// Mitsubishi GX Works2 project: PLC 특수기능 (래치 릴레이)   PLC: Q03UDV

PROGRAM MAIN
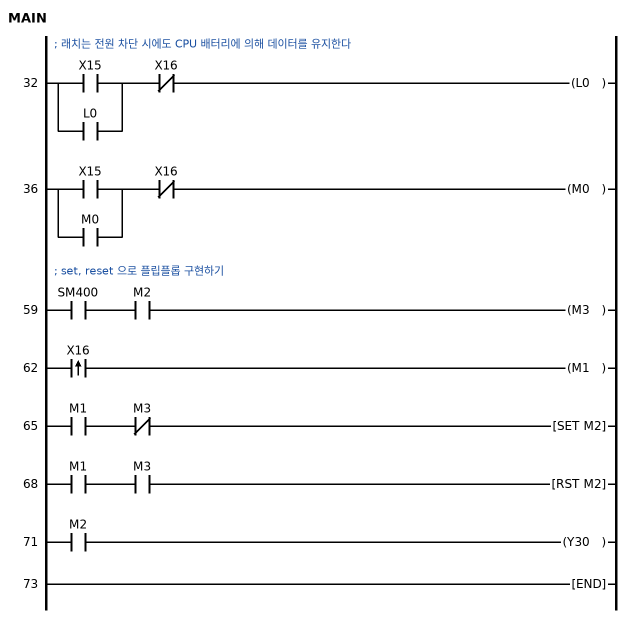
; 래치는 전원 차단 시에도 CPU 배터리에 의해 데이터를 유지한다
32    LD      X15
      OR      L0
      ANI     X16
      OUT     L0
36    LD      X15
      OR      M0
      ANI     X16
      OUT     M0
; set, reset 으로 플립플롭 구현하기
59    LD      SM400
      AND     M2
      OUT     M3
62    LDP     X16
      OUT     M1
65    LD      M1
      ANI     M3
      SET     M2
68    LD      M1
      AND     M3
      RST     M2
71    LD      M2
      OUT     Y30
73    END
END_PROGRAM
